(* IEC 61131-3 sources: Codesys_MELSEC_Comm_Sample/src, 2 files *)

(* ---- PLC_PRG_Example1.st ---- *)
PROGRAM PLC_PRG_Example1
VAR
    fbReadWord    : FB_SlmpReadWordService;
    fbWriteWord   : FB_SlmpWriteWordService;
    fbReadBit     : FB_SlmpReadBitService;
    fbWriteBit    : FB_SlmpWriteBitService;
    fbReadPlcInfo : FB_SlmpReadPlcInfoService;
    fbCloseAll    : FB_SlmpCloseConnection;

    // Pulse these from HMI/debug (1-scan ON recommended)
    xTrigReadWord    : BOOL := FALSE;
    xTrigWriteWord   : BOOL := FALSE;
    xTrigReadBit     : BOOL := FALSE;
    xTrigWriteBit    : BOOL := FALSE;
    xTrigReadPlcInfo : BOOL := FALSE;
    xTrigCloseAll    : BOOL := FALSE;

    // Connection settings (PLC1)
    sTargetIp      : STRING := '192.168.3.10';
    uiTargetPort   : UINT := 4001;
    xUse4EFrame    : BOOL := TRUE;
    xUseUdpFrame   : BOOL := TRUE; // FALSE: TCP, TRUE: UDP
    uiFrameSerialNo: UINT := 1;

    // Write buffers
    aWriteWords : ARRAY[0..SLMP_MAX_WORD_INDEX] OF UINT;
    aWriteBits  : ARRAY[0..SLMP_MAX_BIT_INDEX] OF BOOL;

    // Monitor outputs
    xReadWordDone    : BOOL;
    xWriteWordDone   : BOOL;
    xReadBitDone     : BOOL;
    xWriteBitDone    : BOOL;
    xReadPlcInfoDone : BOOL;

    uiWordRead0 : UINT;
    uiWordRead1 : UINT;
    xBitRead0   : BOOL;
    xBitRead1   : BOOL;
    xBitRead2   : BOOL;
    xBitRead3   : BOOL;

    uiPlcTypeCodeMon : UINT;
    xPlcRunMon       : BOOL;
    xPlcStopMon      : BOOL;
    uiPlcModeMon     : UINT;
    sPlcTypeNameMon  : STRING(16);

    sLastErrorText : STRING;
END_VAR

// === IMPLEMENTATION ===
// Example write data
aWriteWords[0] := 16#1234;
aWriteWords[1] := 16#5678;

aWriteBits[0] := TRUE;
aWriteBits[1] := FALSE;
aWriteBits[2] := TRUE;
aWriteBits[3] := TRUE;
aWriteBits[4] := FALSE;
aWriteBits[5] := FALSE;
aWriteBits[6] := TRUE;
aWriteBits[7] := FALSE;

fbReadWord(
    xExecute := xTrigReadWord,
    sIp := sTargetIp,
    uiPort := uiTargetPort,
    udiHeadDevNo := 100,
    uiDeviceCode := SLMP_DEV_D,
    uiPoints := 4,
    tTimeout := T#2S,
    uiRetryMax := 2,
    tReconnectDelay := T#500MS,
    xUse4E := xUse4EFrame,
    xUseUdp := xUseUdpFrame,
    uiSerialNo := uiFrameSerialNo
);

fbWriteWord(
    xExecute := xTrigWriteWord,
    sIp := sTargetIp,
    uiPort := uiTargetPort,
    udiHeadDevNo := 200,
    uiDeviceCode := SLMP_DEV_D,
    uiPoints := 2,
    tTimeout := T#2S,
    uiRetryMax := 2,
    tReconnectDelay := T#500MS,
    xUse4E := xUse4EFrame,
    xUseUdp := xUseUdpFrame,
    uiSerialNo := uiFrameSerialNo,
    aWriteValues := aWriteWords
);

fbReadBit(
    xExecute := xTrigReadBit,
    sIp := sTargetIp,
    uiPort := uiTargetPort,
    udiHeadDevNo := 1000,
    uiDeviceCode := SLMP_DEV_M,
    uiPoints := 8,
    tTimeout := T#2S,
    uiRetryMax := 2,
    tReconnectDelay := T#500MS,
    xUse4E := xUse4EFrame,
    xUseUdp := xUseUdpFrame,
    uiSerialNo := uiFrameSerialNo
);

fbWriteBit(
    xExecute := xTrigWriteBit,
    sIp := sTargetIp,
    uiPort := uiTargetPort,
    udiHeadDevNo := 1000,
    uiDeviceCode := SLMP_DEV_M,
    uiPoints := 8,
    tTimeout := T#2S,
    uiRetryMax := 2,
    tReconnectDelay := T#500MS,
    xUse4E := xUse4EFrame,
    xUseUdp := xUseUdpFrame,
    uiSerialNo := uiFrameSerialNo,
    aWriteBits := aWriteBits
);

fbReadPlcInfo(
    xExecute := xTrigReadPlcInfo,
    sIp := sTargetIp,
    uiPort := uiTargetPort,
    tTimeout := T#2S,
    uiRetryMax := 2,
    tReconnectDelay := T#500MS,
    xUse4E := xUse4EFrame,
    xUseUdp := xUseUdpFrame,
    uiSerialNo := uiFrameSerialNo
);

fbCloseAll(
    xExecute := xTrigCloseAll
);

xReadWordDone := fbReadWord.xDone;
xWriteWordDone := fbWriteWord.xDone;
xReadBitDone := fbReadBit.xDone;
xWriteBitDone := fbWriteBit.xDone;
xReadPlcInfoDone := fbReadPlcInfo.xDone;

uiWordRead0 := fbReadWord.aReadValues[0];
uiWordRead1 := fbReadWord.aReadValues[1];
xBitRead0 := fbReadBit.aReadBits[0];
xBitRead1 := fbReadBit.aReadBits[1];
xBitRead2 := fbReadBit.aReadBits[2];
xBitRead3 := fbReadBit.aReadBits[3];
uiPlcTypeCodeMon := fbReadPlcInfo.uiPlcTypeCode;
xPlcRunMon := fbReadPlcInfo.xPlcRun;
xPlcStopMon := fbReadPlcInfo.xPlcStop;
uiPlcModeMon := fbReadPlcInfo.uiPlcMode;
sPlcTypeNameMon := fbReadPlcInfo.sPlcTypeName;

IF fbReadWord.xError THEN
    IF fbReadWord.diError >= 0 THEN
        sLastErrorText := F_SlmpEndCodeText(uiEndCode := TO_UINT(fbReadWord.diError));
    ELSE
        sLastErrorText := 'LOCAL_ERROR';
    END_IF;
ELSIF fbWriteWord.xError THEN
    IF fbWriteWord.diError >= 0 THEN
        sLastErrorText := F_SlmpEndCodeText(uiEndCode := TO_UINT(fbWriteWord.diError));
    ELSE
        sLastErrorText := 'LOCAL_ERROR';
    END_IF;
ELSIF fbReadBit.xError THEN
    IF fbReadBit.diError >= 0 THEN
        sLastErrorText := F_SlmpEndCodeText(uiEndCode := TO_UINT(fbReadBit.diError));
    ELSE
        sLastErrorText := 'LOCAL_ERROR';
    END_IF;
ELSIF fbWriteBit.xError THEN
    IF fbWriteBit.diError >= 0 THEN
        sLastErrorText := F_SlmpEndCodeText(uiEndCode := TO_UINT(fbWriteBit.diError));
    ELSE
        sLastErrorText := 'LOCAL_ERROR';
    END_IF;
ELSIF fbReadPlcInfo.xError THEN
    IF fbReadPlcInfo.diError >= 0 THEN
        sLastErrorText := F_SlmpEndCodeText(uiEndCode := TO_UINT(fbReadPlcInfo.diError));
    ELSE
        sLastErrorText := 'LOCAL_ERROR';
    END_IF;
END_IF;

(* ---- PLC_PRG_Example2.st ---- *)
PROGRAM PLC_PRG_Example
VAR
    fbWriteWordPlc1 : FB_SlmpWriteWordService;
    fbWriteWordPlc2 : FB_SlmpWriteWordService;
    fbWriteWordPlc3 : FB_SlmpWriteWordService;
    fbWriteWordPlc4 : FB_SlmpWriteWordService;

    xEnableWritePlc1 : BOOL := TRUE;
    xEnableWritePlc2 : BOOL := TRUE;
    xEnableWritePlc3 : BOOL := TRUE;
    xEnableWritePlc4 : BOOL := TRUE;

    xTrigWritePlc1 : BOOL;
    xTrigWritePlc2 : BOOL;
    xTrigWritePlc3 : BOOL;
    xTrigWritePlc4 : BOOL;

    xWriteBusyPlc1 : BOOL;
    xWriteBusyPlc2 : BOOL;
    xWriteBusyPlc3 : BOOL;
    xWriteBusyPlc4 : BOOL;

    xWriteDonePlc1 : BOOL;
    xWriteDonePlc2 : BOOL;
    xWriteDonePlc3 : BOOL;
    xWriteDonePlc4 : BOOL;

    xWriteErrorPlc1 : BOOL;
    xWriteErrorPlc2 : BOOL;
    xWriteErrorPlc3 : BOOL;
    xWriteErrorPlc4 : BOOL;

    diWriteErrorPlc1 : DINT;
    diWriteErrorPlc2 : DINT;
    diWriteErrorPlc3 : DINT;
    diWriteErrorPlc4 : DINT;

    sLastErrorText  : STRING;

    sTargetIpPlc1    : STRING := '192.168.3.10';
    uiTargetPortPlc1 : UINT := 4001;
    sTargetIpPlc2    : STRING := '192.168.3.11';
    uiTargetPortPlc2 : UINT := 4001;
    sTargetIpPlc3    : STRING := '192.168.3.12';
    uiTargetPortPlc3 : UINT := 4001;
    sTargetIpPlc4    : STRING := '192.168.3.13';
    uiTargetPortPlc4 : UINT := 4001;

    xUse4EFrame      : BOOL := TRUE;
    xUseUdpFrame     : BOOL := TRUE; // FALSE: TCP, TRUE: UDP
    uiFrameSerialNo  : UINT := 1;

    aWriteWords      : ARRAY[0..SLMP_MAX_WORD_INDEX] OF UINT;
    udRandState      : UDINT := 16#12345678;
    uiIdx            : UINT;
END_VAR

// === IMPLEMENTATION ===
// Generate random data for 100 words (D0..D99) every scan.
FOR uiIdx := 0 TO 99 DO
    udRandState := udRandState * 1664525 + 1013904223;
    aWriteWords[uiIdx] := TO_UINT(udRandState AND 16#0000FFFF);
END_FOR;

// Do not retrigger while busy. Re-run after done or error.
xTrigWritePlc1 := xEnableWritePlc1 AND (NOT fbWriteWordPlc1.xBusy);
xTrigWritePlc2 := xEnableWritePlc2 AND (NOT fbWriteWordPlc2.xBusy);
xTrigWritePlc3 := xEnableWritePlc3 AND (NOT fbWriteWordPlc3.xBusy);
xTrigWritePlc4 := xEnableWritePlc4 AND (NOT fbWriteWordPlc4.xBusy);

fbWriteWordPlc1(
    xExecute := xTrigWritePlc1,
    sIp := sTargetIpPlc1,
    uiPort := uiTargetPortPlc1,
    udiHeadDevNo := 0,
    uiDeviceCode := SLMP_DEV_D,
    uiPoints := 100,
    tTimeout := T#2S,
    uiRetryMax := 2,
    tReconnectDelay := T#500MS,
    xUse4E := xUse4EFrame,
    xUseUdp := xUseUdpFrame,
    uiSerialNo := uiFrameSerialNo,
    aWriteValues := aWriteWords
);

fbWriteWordPlc2(
    xExecute := xTrigWritePlc2,
    sIp := sTargetIpPlc2,
    uiPort := uiTargetPortPlc2,
    udiHeadDevNo := 0,
    uiDeviceCode := SLMP_DEV_D,
    uiPoints := 100,
    tTimeout := T#2S,
    uiRetryMax := 2,
    tReconnectDelay := T#500MS,
    xUse4E := xUse4EFrame,
    xUseUdp := xUseUdpFrame,
    uiSerialNo := uiFrameSerialNo,
    aWriteValues := aWriteWords
);

fbWriteWordPlc3(
    xExecute := xTrigWritePlc3,
    sIp := sTargetIpPlc3,
    uiPort := uiTargetPortPlc3,
    udiHeadDevNo := 0,
    uiDeviceCode := SLMP_DEV_D,
    uiPoints := 100,
    tTimeout := T#2S,
    uiRetryMax := 2,
    tReconnectDelay := T#500MS,
    xUse4E := xUse4EFrame,
    xUseUdp := xUseUdpFrame,
    uiSerialNo := uiFrameSerialNo,
    aWriteValues := aWriteWords
);

fbWriteWordPlc4(
    xExecute := xTrigWritePlc4,
    sIp := sTargetIpPlc4,
    uiPort := uiTargetPortPlc4,
    udiHeadDevNo := 0,
    uiDeviceCode := SLMP_DEV_D,
    uiPoints := 100,
    tTimeout := T#2S,
    uiRetryMax := 2,
    tReconnectDelay := T#500MS,
    xUse4E := xUse4EFrame,
    xUseUdp := xUseUdpFrame,
    uiSerialNo := uiFrameSerialNo,
    aWriteValues := aWriteWords
);

xWriteBusyPlc1 := fbWriteWordPlc1.xBusy;
xWriteBusyPlc2 := fbWriteWordPlc2.xBusy;
xWriteBusyPlc3 := fbWriteWordPlc3.xBusy;
xWriteBusyPlc4 := fbWriteWordPlc4.xBusy;

xWriteDonePlc1 := fbWriteWordPlc1.xDone;
xWriteDonePlc2 := fbWriteWordPlc2.xDone;
xWriteDonePlc3 := fbWriteWordPlc3.xDone;
xWriteDonePlc4 := fbWriteWordPlc4.xDone;

xWriteErrorPlc1 := fbWriteWordPlc1.xError;
xWriteErrorPlc2 := fbWriteWordPlc2.xError;
xWriteErrorPlc3 := fbWriteWordPlc3.xError;
xWriteErrorPlc4 := fbWriteWordPlc4.xError;

diWriteErrorPlc1 := fbWriteWordPlc1.diError;
diWriteErrorPlc2 := fbWriteWordPlc2.diError;
diWriteErrorPlc3 := fbWriteWordPlc3.diError;
diWriteErrorPlc4 := fbWriteWordPlc4.diError;

IF xWriteErrorPlc1 THEN
    IF diWriteErrorPlc1 >= 0 THEN
        sLastErrorText := F_SlmpEndCodeText(uiEndCode := TO_UINT(diWriteErrorPlc1));
    ELSE
        sLastErrorText := 'LOCAL_ERROR';
    END_IF;
ELSIF xWriteErrorPlc2 THEN
    IF diWriteErrorPlc2 >= 0 THEN
        sLastErrorText := F_SlmpEndCodeText(uiEndCode := TO_UINT(diWriteErrorPlc2));
    ELSE
        sLastErrorText := 'LOCAL_ERROR';
    END_IF;
ELSIF xWriteErrorPlc3 THEN
    IF diWriteErrorPlc3 >= 0 THEN
        sLastErrorText := F_SlmpEndCodeText(uiEndCode := TO_UINT(diWriteErrorPlc3));
    ELSE
        sLastErrorText := 'LOCAL_ERROR';
    END_IF;
ELSIF xWriteErrorPlc4 THEN
    IF diWriteErrorPlc4 >= 0 THEN
        sLastErrorText := F_SlmpEndCodeText(uiEndCode := TO_UINT(diWriteErrorPlc4));
    ELSE
        sLastErrorText := 'LOCAL_ERROR';
    END_IF;
END_IF;
